// TIA Portal V15.1 export
// export: Created 2020-06-12T07:35:54.3974609Z, ExportSetting None, DisplayName Totally Integrated Automation Portal, DisplayVersion V15.1, DisplayName TIA Portal Openness, DisplayVersion V15.1, DisplayName STEP 7 Professional, DisplayVersion V15.1, DisplayName STEP 7 Safety, DisplayVersion V15.1, DisplayName WinCC Advanced, DisplayVersion V15.1
FUNCTION "Desk_ES1YD01" : Void   // FC164, FBD
{ S7_Optimized_Access := 'TRUE' }
// stored: SetENOAutomatically False
BEGIN

REGION Network 1: Access door ES1YD01 control
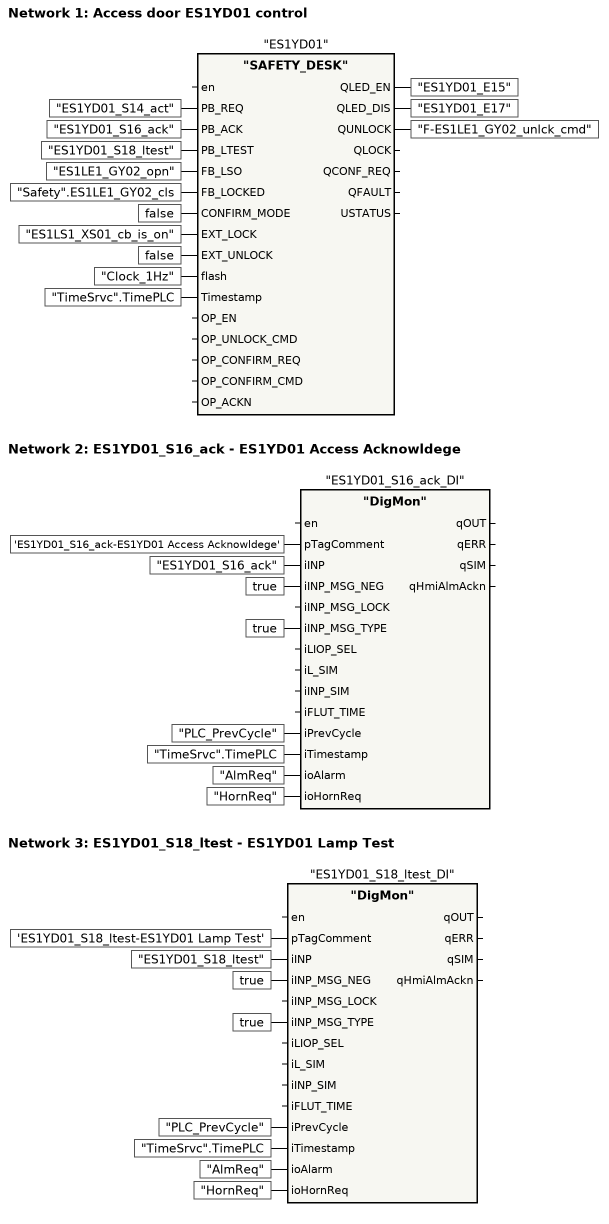
   "ES1YD01"(PB_REQ := "ES1YD01_S14_act",   // "SAFETY_DESK"
             PB_ACK := "ES1YD01_S16_ack",
             PB_LTEST := "ES1YD01_S18_ltest",
             FB_LSO := "ES1LE1_GY02_opn",
             FB_LOCKED := "Safety".ES1LE1_GY02_cls,
             CONFIRM_MODE := false,
             EXT_LOCK := "ES1LS1_XS01_cb_is_on",
             EXT_UNLOCK := false,
             flash := "Clock_1Hz",
             Timestamp := "TimeSrvc".TimePLC,
             QLED_EN => "ES1YD01_E15",
             QLED_DIS => "ES1YD01_E17",
             QUNLOCK => "F-ES1LE1_GY02_unlck_cmd");
END_REGION

REGION Network 2: ES1YD01_S16_ack - ES1YD01 Access Acknowldege
   "ES1YD01_S16_ack_DI"(pTagComment := 'ES1YD01_S16_ack-ES1YD01 Access Acknowldege',   // "DigMon"
                        iINP := "ES1YD01_S16_ack",
                        iINP_MSG_NEG := true,
                        iINP_MSG_TYPE := true,
                        iPrevCycle := "PLC_PrevCycle",
                        iTimestamp := "TimeSrvc".TimePLC,
                        ioAlarm := "AlmReq",
                        ioHornReq := "HornReq");
END_REGION

REGION Network 3: ES1YD01_S18_ltest - ES1YD01 Lamp Test
   "ES1YD01_S18_ltest_DI"(pTagComment := 'ES1YD01_S18_ltest-ES1YD01 Lamp Test',   // "DigMon"
                          iINP := "ES1YD01_S18_ltest",
                          iINP_MSG_NEG := true,
                          iINP_MSG_TYPE := true,
                          iPrevCycle := "PLC_PrevCycle",
                          iTimestamp := "TimeSrvc".TimePLC,
                          ioAlarm := "AlmReq",
                          ioHornReq := "HornReq");
END_REGION

REGION Network 4: ES1YD01_S14_act - ES1YD01 Access Request
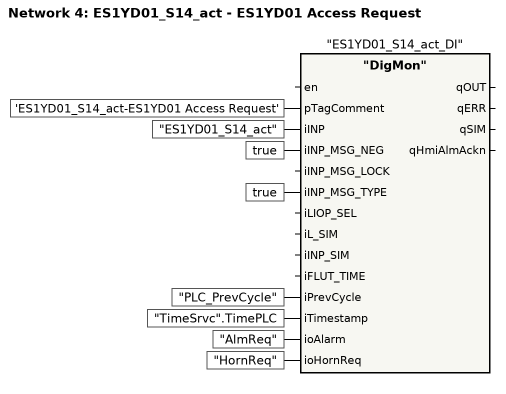
   "ES1YD01_S14_act_DI"(pTagComment := 'ES1YD01_S14_act-ES1YD01 Access Request',   // "DigMon"
                        iINP := "ES1YD01_S14_act",
                        iINP_MSG_NEG := true,
                        iINP_MSG_TYPE := true,
                        iPrevCycle := "PLC_PrevCycle",
                        iTimestamp := "TimeSrvc".TimePLC,
                        ioAlarm := "AlmReq",
                        ioHornReq := "HornReq");
END_REGION
END_FUNCTION
